# EPICS StreamDevice protocol: smb100a-local/smb100aApp/Db/smb100a.proto
# smb100a.proto for DMB100A Signal Generator
Terminator = LF;

get_id {
   out "*idn?";
   in "%#s";
}

get_freq {
   out "freq?"
   in "%f"
}

get_outp {
   out "outp?"
   in "%d"
}

get_out_pwr {
   out "pow?"
   in "%f"
}
